	ADL AT %M*				: REAL := 1.0;		//Gräns konfliktlarm~wp:[unit]%
	AD AT %M*		 		: INT := 60;		//Larmfördröjning konfliktlarm~wp:[unit]s
END_VAR

	//Blockering handställning
	IF bInterlock THEN
		M := FALSE;
	END_IF;

	//Handställning
	IF M  THEN
		OP := OPM; 
	ELSE
		OP := rSetpoint;  
	END_IF
	
	//Handställningslarm
	fbAlarm2(bInput:=M , tAlarmDelay:= , bAutoReset:=TRUE , bAlarmOutput=>AL8 );
	
	//Invertering utång
	IF bInvert THEN
		rOutputInternal := (100 - OP);
	ELSE 
		rOutputInternal := OP;
	END_IF;		
		
	//Hantering utgång	
	FB_BA_AO01(
		rX:= rOutputInternal, 
		rX01:= 0, 
		rX02:= 100, 
		rY01:= 0, 
		rY02:= 32767 , 
		udiOpMod:= , 
		rXManual:= , 
		rY=> rY, 
		TO_iY=>TO_iY );
		
	//Hantering ingång (för feedback)
		FB_BA_AI01(
	TI_usiState:= usiState, 
	TI_iDataIn:= iDataIn, 
	eTerminal:= AIiBusTermType, 
	eSensor:= 0, (* 0 = pt1000, *)
	bConfigurate:= , 
	rX01:=AIrScaleX1 , 
	rX02:=AIrScaleX2 , 
	rY01:= AIrScaleMin, 
	rY02:= AIrScaleMax, 
	rOffset:= , 
	rSmoothingFactor:= , 
	udiDecimalPlace:= , 
	bEnLimitCtrl:= , 
	rHighLimit:= , 
	rLowLimit:=, 
	udiDelayLimitCtrl_sec:= , 
	TO_usiCtrl=> usiCtrl, 
	TO_iDataOut=> iDataOut, 
	rVal=> , 
	bWireBreak=> , 
	bShortCircuit=> , 
	bHighLimit=> , 
	bLowLimit=> , 
	bErr=> , 
	sErrDescr=> );
	
	FB_BA_TiAvrg01(
	bEn:= TRUE, 
	bEnAvrg := TRUE,
	lrIn:=REAL_TO_LREAL(FB_BA_AI01.rVal), 
	udiIntval:=1, 
	udiNumOfElem:= iMedelvardeSekunder, 
	lrOut=> );
	
	IF AI_M THEN
		PV := AI_OPM;
	ELSE
		PV := LREAL_TO_REAL(FB_BA_TiAvrg01.lrOut) + rCal;
	END_IF
	
FAULT := FB_BA_AI01.bWireBreak OR FB_BA_AI01.bShortCircuit;

//Konfliktlarm återföring; tillåt larmtimer om OP ej förändrats mer än tillåten avvikelse, larmvillkor om avvikelse OP-PV större än gräns
IF ABS(OP - rOPold) > ADL THEN
	fbAlarmFb.bInput := FALSE;
	rOPold := OP;
ELSE
	fbAlarmFb.bInput:= ABS(OP - PV) > ADL;
END_IF

fbAlarmFb(tAlarmDelay:= DINT_TO_TIME(AD) * 1000, bAutoReset:=TRUE , bAlarmOutput=>AL );

END_FUNCTION_BLOCK

// oaksLibrary/Utsignal DO_AO/fbComfoVent
//Hantering av vädringsluckor som är pulstidsstyrda med öppetindikering (ej stängt)
FUNCTION_BLOCK fbComfoVent
VAR_INPUT
	V1 AT %M*	: BOOL; //Kommando öppna läge 1 (delvis öppet) ~wp:[trendoptions]i:14400, t:1
	V2 AT %M*	: BOOL; //Kommando öppna läge 2 (fullt öppet) ~wp:[trendoptions]i:14400, t:1
	bInd : BOOL; //Öppetindikering;
END_VAR
VAR_OUTPUT
	bOppna	: BOOL; //Kommando öppna (till DO)
	bStang	: BOOL; //Kommando stäng (till DO)
	PV1 AT %M* : STRING(30); //Aktuellt läge ~wp:
	AL AT %M*	: BOOL; //Fel läge vädringsluckor~wp:
	AL8 AT %M* : BOOL; //Vädringsluckor ej i autoläge ~wp:
END_VAR
VAR
	fbPuls	: TON;
	bInit : BOOL := TRUE;
	
	fbEdge1, fbEdge2 : fbEdge;
	fbAlarm : fbAlarm;
	bStangInt : BOOL;
END_VAR

VAR_INPUT PERSISTENT
	SP1 AT %M* : UINT := 15; //Gångtid kommando läge 1 (delvis öppet) ~wp:[unit]s
	SP2 AT %M* : UINT := 30; //Gångtid kommando läge 2 (fullt  öppet) ~wp:[unit]s
	SP3 AT %M* : UINT := 40; //Gångtid kommando stängt~wp:[unit]s
	AD AT %M*	: UINT := 120; //Fördröjning larm fel läge~wp:[unit]s
	MCMD AT %M* : BYTE; //Handkörning (Auto, Stäng, Öppna delvis, Öppna helt)~wp:[trendoptions]i:14400, t:1
END_VAR

//Handkörning: 1 = Stäng, 2 = Öppna delvis, 3 = Öppna helt
IF MCMD = 1 THEN
	V1 := FALSE;
	V2 := FALSE;
ELSIF MCMD = 2 THEN
	V1 := TRUE;
	V2 := FALSE;
ELSIF MCMD = 3 THEN
	V1 := FALSE;
	V2 := TRUE;
END_IF

AL8 := MCMD <> 0;

//Kolla om något av ingående kommandon förändrats
fbEdge1(anyInput := V1);
fbEdge2(anyInput := V2);

fbPuls.IN := FALSE;

//Återställ puls
IF fbEdge1.bEdgeF OR fbEdge2.bEdgeF THEN
	fbPuls(IN := FALSE);
END_IF

//Om kommando förändrats eller vid uppstart, börja alltid med att stänga helt för att få stängt läge som utgångspunkt
IF fbEdge1.bEdgeSR OR fbEdge2.bEdgeSR OR bInit OR bStangInt THEN
	fbPuls.PT := UINT_TO_TIME(SP3) * 1000;
	fbPuls.IN := TRUE;
	bOppna := FALSE;
	bStang := NOT fbPuls.Q;
	
	IF fbPuls.Q AND NOT bInd THEN
		fbEdge1(bRst := TRUE);
		fbEdge2(bRst := TRUE);
		bInit := FALSE; 
		bStangInt := FALSE;
		fbPuls.IN := FALSE;
	END_IF
	
ELSE
	//Öppna delvis
	IF V1 THEN
		fbPuls.IN := TRUE;
		fbPuls.PT := UINT_TO_TIME(SP1) * 1000;
		bOppna := NOT fbPuls.Q;
	//Öppna helt 
	ELSIF V2 THEN
		fbPuls.IN := TRUE;
		fbPuls.PT := UINT_TO_TIME(SP2) * 1000;
		bOppna := NOT fbPuls.Q;
	END_IF;
END_IF;

fbPuls();

//Larm fel läge
fbAlarm(bInput := (V1 OR V2) XOR bInd, tAlarmDelay := DINT_TO_TIME(AD) * 1000, bAutoReset := TRUE, bAlarmOutput => AL);

//Sätt statustext
IF bStang THEN
	PV1 := 'Stänger';
ELSIF bOppna THEN
	PV1 := 'Öppnar';
ELSIF NOT (V1 OR V2) THEN
	PV1 := 'Stängt';
ELSIF V1 THEN
	PV1 := 'Delvis öppet';
ELSIF V2 THEN
	PV1 := 'Helt öppet';
END_IF;

END_FUNCTION_BLOCK

// oaksLibrary/Utsignal DO_AO/fbDigitalSignalLogicFb
//Block för digitala utsignaler med möjlighet att handställa utsignal. Larmar vid handställning.
//Ingång för lägesåterföring (feedback) för visning samt generering av larm om konflikt mellan M och V0/V1 (feedback)
FUNCTION_BLOCK fbDigitalSignalLogicFb
VAR_INPUT
	bStart : BOOL; //startvillkor
	bSafe: BOOL; //Säkerhetsvillkor
	bHandsetBlock : BOOL; //Används för blockering av handställning utan att blockera utsignal i autoläge. OBS! - För säkerhetsvillkor se ingång bSafe!
	tStartDelay : TIME := T#0S; //Startfördröjning
	tStopDelay : TIME := T#0S; //Stoppfördröjning
	
	V0 AT %I* : BOOL; //Indikering stängd~wp:[trendoptions]i:14400, t:1
	V1 AT %I* : BOOL; //Indikering öppen~wp:[trendoptions]i:14400, t:1
END_VAR
VAR_OUTPUT
	{attribute 'OPC.UA.DA' := '1'}
	CMD AT %Q* 			: BOOL; 		//Utsignal~wp:[trendoptions]i:300[trendoptions]i:14400, t:1
	{attribute 'OPC.UA.DA' := '1'}
	AL8 AT %M* 			: BOOL; 		//Utsignal handställd~wp:[alarmoptions]p:3
	STATE1 AT %M* 		: STRING; 		//Status IO-modul~wp:
	tStartDelayRemaining: TIME; 		//Aktuell  återstående tid startfördröjning
	tStopDelayRemaining : TIME; 		//Aktuell återstående tid toppfördröjning
	AL AT %M* 			: BOOL;			//Konfliktlarm~wp:[alarmoptions]p:3
END_VAR
VAR
	bInternalStart 		: BOOL;
	fbAlarm2 			: fbAlarm; //Larm handställning
	fbAlarmFb			: fbAlarm; //Konfliktlarm
	//Handställningsvariabler från IO
	TI_bStateAuto AT %I* 	:BOOL :=TRUE; //Status Auto/Manuell
	TI_bStateRelay AT %I* 	:BOOL :=FALSE; //Status reläutgång
	bIOManual 				: BOOL;
	
	fbStartDelay	: TON; //Startfördröjning
	fbStopDelay		: TOF; //Stoppfördröjning
END_VAR
VAR_INPUT PERSISTENT
	{attribute 'OPC.UA.DA' := '1'}
	M AT %M* 	: BOOL; //Handställning~wp:[trendoptions]i:14400, t:1
	{attribute 'OPC.UA.DA' := '1'}
	MCMD AT %M* : BOOL; //Styrsignal handställning~wp:[trendoptions]i:14400, t:1
	
	AD AT %M* 	: INT := 60; //Larmfördröjning konfliktlarm~wp:[unit]s
END_VAR

	//Handställning
	fbAlarm2(bInput:=M OR NOT TI_bStateAuto, tAlarmDelay:= , bAutoReset:=TRUE , bAlarmOutput=>AL8 );
	
	IF NOT bSafe OR bHandsetBlock THEN
		M := FALSE;
	END_IF;
	
	//Manuell omkopplare IO-modul
	bIOManual := fKx2652State(bAuto := TI_bStateAuto, bRelayStatus := TI_bStateRelay, sState => STATE1);
	
	
	//Start-/stoppfördröjning
    fbStartDelay(IN:=bStart , PT:=tStartDelay , Q=> , ET=> );
	fbStopDelay(IN:=fbStartDelay.Q, PT:=tStopDelay , Q=> , ET=> );
	
	tStopDelayRemaining := mTimeRemainingTof(fbStopDelay);
	tStartDelayRemaining := mTimeRemainingTon(fbStartDelay);
	
	bInternalStart := fbStopDelay.Q;
	
	IF NOT TI_bStateAuto THEN
		CMD := bIOManual;
	ELSE
		CMD := (((bInternalStart AND NOT M) OR (M AND MCMD)) AND bSafe) OR bIOManual;
	END_IF
	
//Konfliktlarm återföring
fbAlarmFb(
	bInput:= (CMD AND NOT V1) OR (CMD AND V0) OR (NOT CMD AND V1) OR (NOT CMD AND NOT V0), 
	tAlarmDelay:= DINT_TO_TIME(AD) * 1000, 
	bAutoReset:=TRUE, 
	bAlarmOutput=>AL
);

METHOD PUBLIC mStartDelayRemaining : STRING
VAR_INPUT
	sStatusString : STRING;
END_VAR
VAR
	tTime : TIME; 
END_VAR
	tTime := mTimeRemainingTon(fbStartDelay);
	
	
	IF tTime > T#0S AND tTime < fbStartDelay.PT AND NOT M AND TI_bStateAuto  THEN
 		mStartDelayRemaining := CONCAT(sStatusString,CONCAT(INT_TO_STRING(TIME_TO_INT(tTime/1000)), ' s'));
	ELSE
		mStartDelayRemaining := ' ';
	END_IF
END_METHOD

METHOD PUBLIC mStopDelayRemaining : STRING
VAR_INPUT
	sStatusString : STRING;
END_VAR
VAR
	tTime : TIME; 
END_VAR
	tTime := mTimeRemainingTof(fbStopDelay);
	
	
	IF tTime > T#0S AND tTime < fbStopDelay.PT AND NOT M AND TI_bStateAuto  THEN
 		mStopDelayRemaining := CONCAT(sStatusString,CONCAT(INT_TO_STRING(TIME_TO_INT(tTime/1000)), ' s'));
	ELSE
		mStopDelayRemaining := ' ';
	END_IF
END_METHOD

METHOD PROTECTED mTimeRemainingTof : TIME
VAR_IN_OUT
	fbTof : TOF;
END_VAR
mTimeRemainingTof := fbTof.PT - fbTof.ET;
END_METHOD

METHOD PROTECTED mTimeRemainingTon : TIME
VAR_IN_OUT
	fbTon : TON;
END_VAR
mTimeRemainingTon := fbTon.PT - fbTon.ET;
END_METHOD

END_FUNCTION_BLOCK

// oaksLibrary/Utsignal DO_AO/fbGeneralSignalLogic
//OAKS AB
//2022-10-28
//Generellt analog ut block med handställningsmöjlighet för tex. ventilställdon via SX:Acura
FUNCTION_BLOCK fbGeneralSignalLogic
VAR_INPUT
	rSetpoint 				: REAL := 0; //Skalad insignal för auto-läge (exmepelvis regulatorsignal)
	bInterlock 				: BOOL := FALSE; //Blockering av handställning
	bInvert 				: BOOL := FALSE; //Invertering utgång
END_VAR
VAR_OUTPUT
	{attribute 'OPC.UA.DA' := '1'}
	AL8 AT %M* 				: BOOL := FALSE; //Utsignal handställd~wp:[alarmoptions]p:3
	{attribute 'OPC.UA.DA' := '1'}
	OP AT %M* : REAL;  //Utsignal~wp:[unit]%[format]0[trendoptions]i:300
END_VAR
VAR
	rOutputInternal 		: REAL; //Intern signal för invertering/ej invertering
	rOutputConverted		: REAL; //Signal inverterad eller/ej inverterad
	fbAlarm2 				: fbAlarm; //Larm handställning
END_VAR
VAR_INPUT PERSISTENT
	{attribute 'OPC.UA.DA' := '1'}
	M AT %M*				: BOOL;//Handställning~wp:[trendoptions]i:14400, t:1
	{attribute 'OPC.UA.DA' := '1'}
	OPM AT %M* : REAL;//Värde handställning~wp:[unit]%[format]0
END_VAR

	//Blockering handställning
	IF bInterlock THEN
		M := FALSE;
	END_IF;

	//Handställning
	IF M THEN
		rOutputConverted := OPM; 
	ELSE
		rOutputConverted := rSetpoint;  
	END_IF
	
	//Handställningslarm
	fbAlarm2(bInput:=M , tAlarmDelay:= , bAutoReset:=TRUE , bAlarmOutput=>AL8 );
	
	//Invertering utång
	IF bInvert THEN
		rOutputInternal := (100 - rOutputConverted);
	ELSE 
		rOutputInternal := rOutputConverted;
	END_IF;		

	//Utsignal 
	OP := rOutputInternal;

END_FUNCTION_BLOCK

// oaksLibrary/Utsignal DO_AO/fbLightSignalLogic
// Funktionsblock för utebelysning ute. Valbart driftläge för startvillkor mellan Astrour + Tidkanal och enbart Tidkanal.
// ANVÄND EJ bStart då denna skrivs till internt i blocket.
FUNCTION_BLOCK fbLightSignalLogic EXTENDS fbDigitalSignalLogic
VAR_INPUT
	bTidkanal : BOOL; // Koppla tidkanal hit.
	bAstrour : BOOL; // Koppla utgång från fbSunclock hit.
END_VAR
VAR_OUTPUT
END_VAR
VAR
END_VAR
VAR PERSISTENT
	{attribute 'OPC.UA.DA' := '1'}
	SP1 AT %M* : INT; //1 = Astrour + Tidkanal. 0 = Tidkanal~wp:
END_VAR	
VAR_OUTPUT
	{attribute 'OPC.UA.DA' := '1'}
	PV AT %M* : STRING; //Startvillkor~wp:
END_VAR

SUPER^();
bStart := mBelysningsvillkor(iDriftlage:= SP1, bTidkanal:=bTidkanal , bAstrour:= bAstrour, sAktuelltDriftlage=>PV);

METHOD PRIVATE mBelysningsvillkor : BOOL
VAR_IN_OUT
	iDriftlage : INT; // 1 om belysningsvillkor OCH tidkanal måste vara till. 0 om bara tidkanal måste vara till.
END_VAR
VAR_INPUT
	bTidkanal : BOOL;
	bAstrour : BOOL; // lux-givare under inställt värde
END_VAR
VAR_OUTPUT
	sAktuelltDriftlage : STRING;
END_VAR
IF bTidkanal AND bAstrour THEN
	mBelysningsvillkor := TRUE;
ELSIF bTidkanal AND iDriftlage = 0 THEN
	mBelysningsvillkor := TRUE;
ELSE
	mBelysningsvillkor := FALSE;
END_IF

IF iDriftlage = 1 THEN
	sAktuelltDriftlage := 'Tidkanal och astrour sätter utgång i läge till.';
ELSE
	sAktuelltDriftlage := 'Tidkanal sätter utgång i läge till.';
END_IF

IF iDriftlage > 1 THEN
	iDriftlage := 1; 
END_IF

IF iDriftlage < 0 THEN
	iDriftlage := 0; 
END_IF
END_METHOD

END_FUNCTION_BLOCK

// oaksLibrary/Utsignal DO_AO/fbLightSignalLogicLux
//Oaks AB
//2022-08-17
//Funktionsblock för utebelysning ute. Valbart driftläge för startvillkor mellan Luxgivare + Tidkanal och enbart Tidkanal.
//ANVÄND EJ bStart då denna skrivs till internt i blocket
FUNCTION_BLOCK fbLightSignalLogicLux EXTENDS fbDigitalSignalLogic
VAR_INPUT
	//Koppla tidkanal hit.
	bTidkanal: BOOL;
	//Koppla utgång från LuxLightCon blocket hit eller egen hyst hit.
	bLux: BOOL;
END_VAR
VAR PERSISTENT
	//1 = Luxgivare + Tidkanal. 0 = Tidkanal~wp:
	{attribute 'OPC.UA.DA' := '1'}
	SP1 AT %M*: INT;
END_VAR
VAR_OUTPUT
	//Startvillkor~wp:
	{attribute 'OPC.UA.DA' := '1'}
	PV AT %M*: STRING;
END_VAR

SUPER^();
bStart := mBelysningsvillkor(iDriftlage:= SP1, bTidkanal:=bTidkanal , bLux:= bLux, sAktuelltDriftlage=>PV);

METHOD mBelysningsvillkor : BOOL
VAR_IN_OUT
	/// 1 om belysningsvillkor OCH tidkanal måste vara till. 0 om bara tidkanal måste vara till.
	iDriftlage: INT;
END_VAR
VAR_INPUT
	bTidkanal: BOOL;
	/// lux-givare under inställt värde
	bLux: BOOL;
END_VAR
VAR_OUTPUT
	sAktuelltDriftlage: STRING;
END_VAR
IF bTidkanal AND bLux THEN
	mBelysningsvillkor := TRUE;
ELSIF bTidkanal AND iDriftlage = 0 THEN
	mBelysningsvillkor := TRUE;
ELSE
	mBelysningsvillkor := FALSE;
END_IF

IF iDriftlage = 1 THEN
	sAktuelltDriftlage := 'Tidkanal och luxgivare sätter utgång i läge till.';
ELSE
	sAktuelltDriftlage := 'Tidkanal sätter utgång i läge till.';
END_IF

IF iDriftlage > 1 THEN
	iDriftlage := 1; 
END_IF

IF iDriftlage < 0 THEN
	iDriftlage := 0; 
END_IF
END_METHOD

END_FUNCTION_BLOCK

// oaksLibrary/Växlingsblock/fbDailyToggle
// Block för att växla mellan två bool-outputs. Växling sker intälld tid varje dag.
FUNCTION_BLOCK fbDailyToggle
VAR_INPUT
	{attribute 'OPC.UA.DA' := '1'}
	M AT %M*  : BOOL; //Manuell växling~wp:[trendoptions]i:14400, t:1
END_VAR
VAR_OUTPUT
	{attribute 'OPC.UA.DA' := '1'}
	PV AT %M* : INT; //Aktuellt val~wp:[trendoptions]i:14400, t:1
	bOutput1, bOutput2 : BOOL;
END_VAR
VAR 
	fbDayTrig: R_trig;
	{attribute 'OPC.UA.DA' := '1'}
	PV4 AT %M* : STRING := ' ' ; //Växling sker intälld tid varje dag. Tiden är ställbar mellan 0000-2359.~wp:
	stTime		: tc2_ba.TIMESTRUCT;
	nActualDayCase	: INT;
	nActualHour 	: INT;
	nActualMinute 	: INT;
	
	FB_BA_GetTime01 : tc2_ba.FB_BA_GetTime; 
	FB_BA_ExtTiSt01 : tc2_ba.FB_BA_ExtTiSt;	
	
	nTime : INT; // Internvariabel aktuell tid (nActualHour+nActualMinute)
//	bDay : BOOL; // Internvariabel blir TRUE om inställd dag är lika med aktuell dag
	bTime : BOOL; // Internvariabel blir TRUE om inställd tid är lika med aktuell tid
END_VAR
VAR_INPUT PERSISTENT
//	SP1 AT %M*  : INT:=1; //Dag för växling (-1 = ingen växling 0 = Söndag 1 = Måndag 2 = Tisdag..7 = Söndag~wp:
	{attribute 'OPC.UA.DA' := '1'}
	SP1 AT %M*  : INT:=1000; //Tid för växling (skrivs i format 1200 för 12:00)~wp:
END_VAR

	FB_BA_GetTime01(bEn :=TRUE);	
	stTime := FB_BA_GetTime01.stSysTi;

//	nActualDayCase :=WORD_TO_INT (stTime.wDayOfWeek);
	nActualHour :=WORD_TO_INT (stTime.wHour)*100;
	nActualMinute :=WORD_TO_INT (stTime.wMinute);
	
	nTime := nActualHour+nActualMinute;
	
//	bDay := nActualDayCase = SP1;
	bTime := nTime = SP1;

//	IF SP1 < -1 OR  SP1>7 THEN
//		SP1 := 1;
//	END_IF
	
	IF SP1 < 0 OR  SP1>2359 THEN
		SP1 := 1200;
	END_IF

	IF PV < 1 OR PV > 2  THEN	
		PV := 1;
	END_IF;

	IF bTime OR M THEN
		fbDayTrig(CLK := TRUE);
	ELSE
		fbDayTrig(CLK := FALSE);
	END_IF

	IF fbDayTrig.Q THEN
		IF PV = 1 THEN
			PV := 2;
		ELSE
			PV := 1;
		END_IF
	END_IF
	
	bOutput1 := (PV = 1);
	bOutput2 := (PV = 2);

END_FUNCTION_BLOCK

// oaksLibrary/Växlingsblock/fbMonthlyToggle
// Block för att växla mellan två bool-outputs. Växling sker intälld tid på inställd dag (-1 till 31).
FUNCTION_BLOCK fbMonthlyToggle
VAR_INPUT
	{attribute 'OPC.UA.DA' := '1'}
	M AT %M*  : BOOL; //Manuell växling~wp:[trendoptions]i:14400, t:1
END_VAR
VAR_OUTPUT
	{attribute 'OPC.UA.DA' := '1'}
	PV AT %M* : INT; //Aktuellt val~wp:[trendoptions]i:14400, t:1
	bOutput1, bOutput2 : BOOL;
END_VAR
VAR 
	fbDayTrig: R_trig;
	{attribute 'OPC.UA.DA' := '1'}
	PV4 AT %M* : STRING := ' ' ; //Växling sker intälld tid på inställd dag (1-31). Ställer man in -1 på "Dag för växling" så inaktiveras växlingen. Tänk på att alla månader inte har 31 dagar. Tiden är ställbar mellan 0000-2359.~wp:
	stTime		: tc2_ba.TIMESTRUCT;
	nActualDayCase	: INT;
	nActualHour 	: INT;
	nActualMinute 	: INT;
	
	FB_BA_GetTime01 : tc2_ba.FB_BA_GetTime; 
	FB_BA_ExtTiSt01 : tc2_ba.FB_BA_ExtTiSt;	
	
	nTime : INT; // Internvariabel aktuell tid (nActualHour+nActualMinute)
	bDay : BOOL; // Internvariabel blir TRUE om inställd dag är lika med aktuell dag
	bTime : BOOL; // Internvariabel blir TRUE om inställd tid är lika med aktuell tid
END_VAR
VAR_INPUT PERSISTENT
	{attribute 'OPC.UA.DA' := '1'}
	SP1 AT %M*  : INT:=1; //Dag för växling (1-31)~wp:
	{attribute 'OPC.UA.DA' := '1'}
	SP2 AT %M*  : INT:=1000; //Tid för växling (skrivs i format 1200 för 12:00)~wp:
END_VAR

	FB_BA_GetTime01(bEn :=TRUE);	
	stTime := FB_BA_GetTime01.stSysTi;

	nActualDayCase :=WORD_TO_INT (stTime.wDay);
	nActualHour :=WORD_TO_INT (stTime.wHour)*100;
	nActualMinute :=WORD_TO_INT (stTime.wMinute);
	
	nTime := nActualHour+nActualMinute;
	
	bDay := nActualDayCase = SP1;
	bTime := nTime = SP2;

	IF SP1 < -1 OR  SP1>31 THEN
		SP1 := 1;
	END_IF
	
	IF SP2 < 0 OR  SP2>2359 THEN
		SP2 := 1200;
	END_IF

	IF PV < 1 OR PV > 2  THEN	
		PV := 1;
	END_IF;

	IF (bDay AND bTime) OR M THEN
		fbDayTrig(CLK := TRUE);
	ELSE
		fbDayTrig(CLK := FALSE);
	END_IF

	IF fbDayTrig.Q THEN
		IF PV = 1 THEN
			PV := 2;
		ELSE
			PV := 1;
		END_IF
	END_IF
	
	bOutput1 := (PV = 1);
	bOutput2 := (PV = 2);

END_FUNCTION_BLOCK

// oaksLibrary/Växlingsblock/fbToggleStep
// Toggle-funktion med uppstegning. Togglar abOutput[0..9] (eller max inst.) i sekvens med inställt intervall när bStart är till.
FUNCTION_BLOCK fbToggleStep
VAR_INPUT
	bStart 		: BOOL;
	iMaxStep	: INT := 9;
	tTimeOn 	: TIME := T#10S;
	tTimeOff 	: TIME := T#10S;
	
END_VAR
VAR_OUTPUT
	iStep		: INT := 0;
	abOutput 	: ARRAY[0..9] OF BOOL;
END_VAR
VAR	
	fbTrigger 	: r_trig;
	fbTon1 		: ton;
	fbTof2 		: tof;
	iX			: INT;
END_VAR

IF iMaxStep > 9 THEN
	iMaxStep := 9;
END_IF

IF bStart THEN
	fbTon1(IN:= NOT fbTof2.Q, PT:= tTimeOff , Q=> , ET=> );
	
	IF fbTon1.Q THEN
		fbTrigger(CLK:=TRUE , Q=> );
		fbTof2(IN:=fbTrigger.Q , PT:=tTimeOn , Q=> , ET=> );
	ELSE
		fbTof2(IN:=FALSE , PT:=tTimeOn , Q=> , ET=> );
		fbTrigger(CLK:=FALSE , Q=> );		
	END_IF
	
	IF fbTrigger.Q THEN
		iStep := iStep + 1;
		IF iStep > iMaxStep THEN
			iStep := 0;
		END_IF
	END_IF
	
	FOR iX := 0 TO 9 DO 
		abOutput[iX] := (iStep = iX) AND fbTof2.Q;
	END_FOR;
ELSE
	FOR iX := 0 TO 9 DO 
		abOutput[iX] := FALSE;
	END_FOR;
END_IF
fbTof2();
fbTon1();

END_FUNCTION_BLOCK

// oaksLibrary/Växlingsblock/fbWeeklyToggle
// Block för att växla mellan två bool-outputs. Växling sker intälld tid på inställd veckodag (-1 till 7).
FUNCTION_BLOCK fbWeeklyToggle
VAR_INPUT
	{attribute 'OPC.UA.DA' := '1'}
	M AT %M*  : BOOL; //Manuell växling~wp:[trendoptions]i:14400, t:1
END_VAR
VAR_OUTPUT
	{attribute 'OPC.UA.DA' := '1'}
	PV AT %M* : INT; //Aktuellt val~wp:[trendoptions]i:14400, t:1
	bOutput1, bOutput2 : BOOL;
END_VAR
VAR 
	fbDayTrig: R_trig;
	{attribute 'OPC.UA.DA' := '1'}
	PV4 AT %M* : STRING := ' ' ; //Växling sker intälld tid på inställd veckodag. Ställer man in -1 på "Dag för växling" så inaktiveras växlingen. Tiden är ställbar mellan 0000-2359.~wp:
	stTime		: tc2_ba.TIMESTRUCT;
	nActualDayCase	: INT;
	nActualHour 	: INT;
	nActualMinute 	: INT;
	
	FB_BA_GetTime01 : tc2_ba.FB_BA_GetTime; 
	FB_BA_ExtTiSt01 : tc2_ba.FB_BA_ExtTiSt;	
	
	nTime : INT; // Internvariabel aktuell tid (nActualHour+nActualMinute)
	bDay : BOOL; // Internvariabel blir TRUE om inställd dag är lika med aktuell dag
	bTime : BOOL; // Internvariabel blir TRUE om inställd tid är lika med aktuell tid
END_VAR
VAR_INPUT PERSISTENT
	{attribute 'OPC.UA.DA' := '1'}
	SP1 AT %M*  : INT:=1; //Dag för växling (0 = Söndag 1 = Måndag 2 = Tisdag..7 = Söndag)~wp:
	{attribute 'OPC.UA.DA' := '1'}
	SP2 AT %M*  : INT:=1000; //Tid för växling (skrivs i format 1200 för 12:00)~wp:
END_VAR

	FB_BA_GetTime01(bEn :=TRUE);	
	stTime := FB_BA_GetTime01.stSysTi;

	nActualDayCase :=WORD_TO_INT (stTime.wDayOfWeek);
	nActualHour :=WORD_TO_INT (stTime.wHour)*100;
	nActualMinute :=WORD_TO_INT (stTime.wMinute);
	
	nTime := nActualHour+nActualMinute;
	
	bDay := nActualDayCase = SP1;
	bTime := nTime = SP2;

	IF SP1 < -1 OR  SP1>7 THEN
		SP1 := 1;
	END_IF
	
	IF SP2 < 0 OR  SP2>2359 THEN
		SP2 := 1200;
	END_IF

	IF PV < 1 OR PV > 2  THEN	
		PV := 1;
	END_IF;

	IF (bDay AND bTime) OR M THEN
		fbDayTrig(CLK := TRUE);
	ELSE
		fbDayTrig(CLK := FALSE);
	END_IF

	IF fbDayTrig.Q THEN
		IF PV = 1 THEN
			PV := 2;
		ELSE
			PV := 1;
		END_IF
	END_IF
	
	bOutput1 := (PV = 1);
	bOutput2 := (PV = 2);

END_FUNCTION_BLOCK

// oaksLibrary/fbExcerciseInactiveMotor
FUNCTION_BLOCK fbExcerciseInactiveMotor		//Funktionsblock för att motionera en komponent efter att den ej körts under viss tid
VAR_INPUT
	bRunIndication	: BOOL;		//Ska vara till när komponenten går (t ex driftsvar)
	tInactiveTime	: TIME;		//Tid som skall passera utan att komponenten går till för att motion skall ske
	tExcerciseTime	: TIME;		//Gångtid motionskörning
END_VAR

VAR
	fbTON			: TON;		//Timer som startar motion
	fbTOF			: TOF;		//Timer för motionering
END_VAR

VAR_OUTPUT
	bOutput			: BOOL;		//Motioneringskommando
	tTimeLeftNext	: TIME;		//Tid kvar till nästa motion
	tTimeLeftExc	: TIME;		//Tid kvar motionering
END_VAR

//Kör TON med inställd tid när komponenten inte går
fbTON(IN := NOT bRunIndication, PT := tInactiveTime);

//Kör TOF med inställd tid när TON gått till, dvs motionering ska starta, skriv utsignal
fbTOF(IN := fbTON.Q, PT := tExcerciseTime, Q => bOutput);	

tTimeLeftNext 	:= tInactiveTime - fbTON.ET;
tTimeLeftExc	:= tExcerciseTime - fbTOF.ET;

END_FUNCTION_BLOCK

// oaksLibrary/fbNightCooling
FUNCTION_BLOCK fbNightCooling
// Funktionsblock för nattkyla
// Ändrat av Robert H, 2021-11-23
// Testat 2021-11-23

// V-tagg i detta block knyts till regulator för att blockera eventuell kylsekvens, till inputen bNightCooling i fbVentilationUnit.
VAR
	fbExhTemperatureTON : TON;
	rLocalTemperatureProcessValue : REAL; // Mellanvariabel för temperatur. Vid nattkyla via frånluftstemperatur uppdateras denna enbart vid driftindikering på frånluftsfläkt.
	summerInternal: BOOL;
	bNightCool : BOOL;
	fbTof_StopDelayNC: TOF;
	fbTon_StartDelaySummer: TON;
	fbTof_StopDelaySummer: TOF;
	sTemp : STRING(255);
	rTempUsed : REAL; // Uteluftstemperatur
END_VAR

VAR_INPUT
	bExhfanInd : BOOL; // Vid nattkyla via frånluftstemp knyt frånluftsfläktens indikering.
	bExhtempMode : BOOL; // Aktivera denna för nattkyla via frånluftstemp.
	rSetpoint : REAL; // Börvärde. Knyt det börvärde som används vid normaldrift (exempelvis utekomp eller kaskad).	
	bTimechannel : BOOL; //Dagdrift (knyt outputen bNormalOperation från fbVentilationUnit)	
	rOutdoorTemperature : ANY; //Utetemperatur knyter man inget här används oaksGVL.rOutdoortemp
END_VAR
VAR_INPUT PERSISTENT
	Enable : BOOL := TRUE; // Tillåt nattkyla (knyt t ex _M-tagg eller villkor från annan funktion)
	{attribute 'OPC.UA.DA' := '1'}
	PV AT %M*  : REAL; //Aktuell temperatur~wp:[unit]°C[format]0.0
	{attribute 'OPC.UA.DA' := '1'}
	SP AT %M*  : REAL := 22; //Rumsbörvärde nattkyla (startar 2.5°C över och stoppar 0.5°C under~wp:[unit]°C[format]0.0
	{attribute 'OPC.UA.DA' := '1'}
	SP1 AT %M*  : REAL := 14; //Börvärde tilluft vid nattkyla~wp:[unit]°C[format]0.0
	{attribute 'OPC.UA.DA' := '1'}
	SP2 AT %M*  : REAL := 12; //Mingräns utetemp för nattkyla~wp:[unit]°C[format]0.0
END_VAR

VAR_OUTPUT
	{attribute 'OPC.UA.DA' := '1'}
	V AT %M* : BOOL; //Nattkyla aktiv~wp:[trendoptions]i:14400, t:1
	{attribute 'OPC.UA.DA' := '1'}
	PV4 AT %M*  : BOOL; // Startvillkor rumstemperatur över~wp:[trendoptions]i:14400, t:1
	{attribute 'OPC.UA.DA' := '1'}
	PV5 AT %M* : BOOL; //Utetemperaturvillkor nattkyla~wp:[trendoptions]i:14400, t:1
	{attribute 'OPC.UA.DA' := '1'}
	PV6 AT %M*  : BOOL; // Startvillkor rumstemperatur högre än utetemp~wp:[trendoptions]i:14400, t:1
	{attribute 'OPC.UA.DA' := '1'}
	PV7 AT %M*  : STRING; // Konfiguration nattkyla~wp:
	{attribute 'OPC.UA.DA' := '1'}
	PV8 AT %M*  : STRING; // Konfiguration nattkyla~wp:
	rSetpointOutput : REAL; // Aktuellt börvärde. Knyts till CSP tilluft (använder man våra setpoint-block knyter man denna till rOverrideSetpoint)
END_VAR

//Temp select
	rTempUsed := F_GetTempToUse(rOutdoorTemperature);

	sTemp := 'Nattkyla via: ';
	IF bExhtempMode THEN
		sTemp := CONCAT(sTemp, 'Frånluftstemperatur');
	ELSE
		sTemp := CONCAT(sTemp, 'Rumstemperatur');	
	END_IF
		
	PV7 := sTemp;
	
	sTemp := 'Aktuell nattkyletemperatur: ';
	
	sTemp := CONCAT(sTemp, REAL_TO_STRING(rLocalTemperatureProcessValue));	
	PV8 :=CONCAT(sTemp, ' °C');
	//Summer	
	IF (rTempUsed > SP2) AND Enable THEN
		summerInternal := TRUE;
	ELSIF (rTempUsed < (SP2 - 0.5)) OR NOT Enable THEN
		summerInternal := FALSE;
	END_IF;
	
	//Start/stop delay summer
   	fbTon_StartDelaySummer(IN:= summerInternal, PT:= T#15M, Q=>, ET=> );
	fbTof_StopDelaySummer(IN:= fbTon_StartDelaySummer.Q, PT:= T#5M, Q=>, ET=> );

	PV5 := fbTon_StartDelaySummer.Q OR fbTof_StopDelaySummer.Q;
	
	
	fbExhTemperatureTON(IN:=bExhfanInd , PT:=T#1M , Q=> , ET=> );
	
	IF fbExhTemperatureTON.Q OR NOT bExhtempMode THEN
		rLocalTemperatureProcessValue := PV;
	END_IF;
	
	IF rLocalTemperatureProcessValue > (SP + 2.5) THEN
		PV4 := TRUE;
	ELSIF rLocalTemperatureProcessValue < (SP - 0.5) THEN
		PV4 := FALSE;
	END_IF
	
	IF rTempUsed < (rLocalTemperatureProcessValue - 4.0) THEN
		PV6 := TRUE;
	ELSIF (rLocalTemperatureProcessValue - rTempUsed) < 3.0 THEN
		PV6 := FALSE;
	END_IF
	
	//Start/stop nightcool
	IF PV4 AND PV6 AND PV5 THEN
		bNightCool := TRUE;
	END_IF
	IF NOT PV4 OR NOT PV6 OR NOT PV5 THEN 
		bNightCool := FALSE;
	END_IF
	
	//Start/stop delay		
	fbTof_StopDelayNC(IN:= bNightCool, PT:= T#5M, Q=>, ET=> );
		
	V := fbTof_StopDelayNC.Q AND NOT bTimechannel;
		

	IF V THEN
		rSetpointOutput := SP1;
	ELSE
		rSetpointOutput := rSetpoint;
	END_IF

END_FUNCTION_BLOCK

// oaksLibrary/fbVentilationUnit
// Block för ventilationsaggregat. Förreglar aggregat vid Frysvakt, Driftfel, Brandlarm, Rökdetektorlarm, utlöst automatsäkring eller övriga förreglingar med möjlighet att sätta egen statustext.
// PV1 och PV2 indikerar ventilationsaggregatets aktuella status. 
FUNCTION_BLOCK fbVentilationUnit
VAR_INPUT
	bSequenceStart : BOOL := TRUE; // Vid sekvensstart knyt global variabel oaksgvl.bSekvensstart1-15 hit. Aggregat blockeras från att starta då denna ingång är FALSE.
	bServiceSwitch : BOOL; // Ingång serviceomkopplare
	bTimechannel : BOOL; // Startvillkor tidkanal
	bExtendedOperation : BOOL; // Startvillkor förlängd drift
	bUserDefinedOperation1 : BOOL; // Startvillkor egendefinierad drift
	sUserDefinedOperation1 : STRING :=  ' '; // Statustext vid egendefinierad drift (bUserDefinedOperation1)
	bUserDefinedOperation2 : BOOL; // Startvillkor egendefinierad drift
	sUserDefinedOperation2 : STRING :=  ' '; // Statustext vid egendefinierad drift (bUserDefinedOperation2)
	bNightCooling : BOOL; // Startvillkor nattkyla (används bara för statustext)
	bNightHeating : BOOL; // Startvillkor nattanvärmning (används bara för statustext)
	bCoolRecycling : BOOL; // Ingång kylåtervinning aggregat (används bara för statustext)
	bDefrostingVvx : BOOL; // Ingång avfrostning vvx (används bara för statustext)
	bFiredamperExercise : BOOL; // Stannar aggregatet och visar statustext. Aggregat återgår till drift efteråt. 
(*förreglingar - stänger ner aggregatet samt blockerar handställning *)
	bFreezeAlarm : BOOL; // Frysvakt
	bPumpAlarm : BOOL; // Driftfel pump värme
	bFireAlarm : BOOL; // Brandlarm
	bSmokeAlarm : BOOL; // Rökdetektorlarm
	bFuseAlarm : BOOL; // Förregling utlöst automatsäkring
	bInterlock : BOOL; // Övrig förregling
	sInterlockDescription : STRING :=  ' '; // Beskrivning för övrig förregling. Text visas i statusfält vid utlöst förregling
	bInterlock2 : BOOL; // Övrig förregling
	sInterlock2Description : STRING :=  ' '; // Beskrivning för övrig förregling. Text visas i statusfält vid utlöst förregling
	bInterlock3 : BOOL; // Övrig förregling
	sInterlock3Description : STRING :=  ' '; // Beskrivning för övrig förregling. Text visas i statusfält vid utlöst förregling
	
	tSupfanStartDelay : TIME := T#45S;
	tExhfanStartDelay : TIME := T#45S;
	
	tDamperStopDelay : TIME := T#10S; 	
	tAfterblowStopDelay : TIME := T#0S; // Efterblåsningstid vid elbatteri. Används för att köra tilluftsfläkten i angiven tid efter aggregatsstopp. !! Denna tidsinställning används även som stoppfördröjning för serviceomkopplare !!
	bAfterblowActive : BOOL := TRUE; // Knyt signal som indikerar att elbatteriet är aktivt. Efterblåsning i inställd tid körs om denna är true. Lämnas denna input tom körs efterblåsning alltid i inställd tid. 
	bSupfan_M : BOOL;
	bSupfan_MCMD : BOOL;
	bSupfanAlarm : BOOL;
	
	bExhfan_M : BOOL;
	bExhfan_MCMD : BOOL;
	bExhfanAlarm : BOOL;
END_VAR
VAR_OUTPUT
	bSupfanOutput : BOOL;
	bSupDamperOutput : BOOL;
	bExhfanOutput : BOOL;
	bExhDamperOutput : BOOL;
	
	bNormalOperation : BOOL; // Är till om aggregatet är i normaldrift (tidkanal eller förlängd drift)
	bNightHeatingStatus : BOOL; // Driftstatus nattanvärmning (Används för eventuell spjällstyrning va exempelvis återluft)
	bAfterBlowElectricHeaterStatus : BOOL; // Driftstatus efterblåsning elbatteri (Används för att blockera elbatteri-sekvens i regulator).
	bSafeCon : BOOL; // Säkerhetsvillkor 
	{attribute 'OPC.UA.DA' := '1'}
	PV1 AT %M* : STRING := ''; //Status aggregatsdrift~wp:[trendoptions]i:14400, t:1
	{attribute 'OPC.UA.DA' := '1'}
	PV2 AT %M* : STRING := ''; //Status aggregatsdrift~wp:[trendoptions]i:14400, t:1
	FAULT AT %M* : BOOL; //Larm lång drifttid~wp:[alarmoptions]p:3
END_VAR
VAR
	PV4 AT %M* : STRING; //Status drifttid~wp:[trendoptions]i:14400, t:1
	{attribute 'OPC.UA.DA' := '1'}
	PV9 AT %M* : BOOL; //Aktivt larm (används för portlet)~wp:[trendoptions]i:14400, t:1
	fbNattAnvarmningsFtrig : f_trig; // Blockerar normaldrift så att aggregat startar upp på nytt efter nattanvärmning
	fbNattAnvarmningsTof : TOF; //  Blockerar normaldrift så att aggregat startar upp på nytt efter nattanvärmning 
	fbInterlockAlarm : fbAlarm;
	bStartCon : BOOL; // Internvariabel startvillkor
	bStartConWithoutAfterblow : BOOL; // Internvariabel startvillkor utan efterblåsningsvillkor
	bExhfanCon : BOOL;
	bCrosswiseInterlock : BOOL;  // korsvis förregling
	
	bExhDamperCon : BOOL;
	
	iStartCase : INT;
	
	fbStartDelayExhFan : TON;
	fbStartDelaySupFan : TON;
	fbResetTon: TON;
	
	sTmpPv1 : STRING;
	sTmpPv2 : STRING;
	
	sRemainingTime : STRING;
	iRemainingTime : INT;
	
	bTmpStartSequenceFlag : BOOL; // internvariabel status startsekvens
	
	bExhDamperOutputInternal : BOOL; 
	bSupDamperOutputInternal : BOOL;
	
	bExhDamperOutputInternalTof : TOF; // Frånslagsfördröjning spjäll
	bSupDamperOutputInternalTof : TOF; // Frånslagsfördröjning spjäll
	fbAfterBlowElectricHeaterInternalTof : TOF; // Frånslagsfördröjning tilluftsfläkt vid efterblåsning elbatteri
	bAfterBlowElectricHeater : BOOL;
	
	fbServiceSwitchTOF : TOF;
	
	fbDrifttidsLarmTON : TON; // Larmar om aggregatet varit igång kontinuerligt utan driftstopp.
END_VAR
VAR PERSISTENT
	AD AT %M* : REAL := -1; //Larm om aggr. drifttid sedan senaste stopp > (-1 inaktiv. larm)~wp:[unit]timmar
END_VAR

//Drifttidslarm om aggregatet varit igång konstant i mer än inställd tid. 
mDrifttidslarm();
// Används för Adrians portlet i webport :)
PV9 := bFreezeAlarm OR bPumpAlarm OR bFireAlarm OR bSmokeAlarm OR bFuseAlarm OR bInterlock OR bInterlock2 OR bInterlock3 OR bCrosswiseInterlock;
fbInterlockAlarm(bInput:=bSupfanAlarm OR bExhfanAlarm , tAlarmDelay:= , bAutoReset:=FALSE , bAlarmOutput=> bCrosswiseInterlock);
bNormalOperation := (bTimechannel OR bExtendedOperation OR bUserDefinedOperation1 OR bUserDefinedOperation2) AND bSafeCon;
// Internvariabel för att blockera frånluftsfläkt vid nattanvärmning
bNightHeatingStatus := bNightHeating AND NOT bNormalOperation AND NOT bNightCooling AND bSafeCon;
fbNattAnvarmningsFtrig(CLK := bNightHeatingStatus);
fbNattAnvarmningsTof(IN:= fbNattAnvarmningsFtrig.Q,PT:=T#1S);
// Efterblåsning elbatteri
fbServiceSwitchTOF(IN:= NOT bServiceSwitch, PT:=tAfterblowStopDelay , Q=> , ET=> ); // För att köra efterblåsning vid serviceomkopplare
bStartConWithoutAfterblow := (bTimechannel OR bExtendedOperation OR bNightCooling OR bNightHeating OR bUserDefinedOperation1 OR bUserDefinedOperation2) AND bAfterblowActive AND NOT bFiredamperExercise;
fbAfterBlowElectricHeaterInternalTof(IN:= bStartConWithoutAfterblow , PT:=tAfterblowStopDelay , Q=>bAfterBlowElectricHeater , ET=> );
bAfterBlowElectricHeaterStatus := bAfterBlowElectricHeater AND ((NOT bNightHeating AND NOT bNormalOperation AND NOT bNightCooling) OR (fbServiceSwitchTOF.Q AND NOT fbServiceSwitchTOF.IN)) AND bSafeCon;

bStartCon := bSequenceStart AND (bTimechannel OR bExtendedOperation OR bNightCooling OR bNightHeating OR bUserDefinedOperation1 OR bUserDefinedOperation2 OR bAfterBlowElectricHeaterStatus) AND NOT bFiredamperExercise;
// Förregling samt handställningsförregling av fläktar. Kopplas till bSafe-ingång på fläkt
bSafeCon := NOT fbNattAnvarmningsTof.Q AND NOT bFreezeAlarm AND NOT bPumpAlarm AND NOT bFireAlarm AND NOT bSmokeAlarm AND NOT bFuseAlarm AND NOT bInterlock AND NOT bInterlock2 AND NOT bInterlock3 AND NOT bCrosswiseInterlock AND fbServiceSwitchTOF.Q;
(* Startsekvens - start *)
bExhDamperCon := (bStartCon AND bSafeCon);
(*************************** Utgång frånluftsspjäll ***************************)
bExhDamperOutputInternal := bExhDamperCon OR (bExhfan_M AND bExhfan_MCMD);
IF bNightHeatingStatus THEN
	fbStartDelayExhFan(IN:=bExhDamperCon , PT:=T#0S , Q=> , ET=> );
ELSE
	fbStartDelayExhFan(IN:=bExhDamperCon , PT:=tExhfanStartDelay , Q=> , ET=> );	
END_IF
(*************************** Utgång frånluftsfläkt ***************************)
bExhfanCon := fbStartDelayExhFan.Q AND (bStartCon AND bSafeCon);
bExhfanOutput := bExhfanCon AND NOT bNightHeatingStatus;
(*************************** Utgång tillluftsspjäll ***************************)
bSupDamperOutputInternal := (bExhfanCon AND (bStartCon AND bSafeCon)) OR (bSupfan_M AND bSupfan_MCMD);
fbStartDelaySupFan(IN:= bSupDamperOutputInternal , PT:=tSupfanStartDelay , Q=> , ET=> );
(*************************** Utgång frånluftsfläkt ***************************)
bSupfanOutput := fbStartDelaySupFan.Q AND (bStartCon AND bSafeCon);
(* Startsekvens - slut *)
bExhDamperOutputInternalTof(IN:=bExhDamperOutputInternal , PT:=tDamperStopDelay , Q=>bExhDamperOutput , ET=> );
bSupDamperOutputInternalTof(IN:= bSupDamperOutputInternal, PT:=tDamperStopDelay , Q=>bSupDamperOutput , ET=> );
//Status aggregatsdrift~wp:
IF bTimechannel AND bSafeCon THEN 
	sTmpPv1 := 'Normaldrift';
	bTmpStartSequenceFlag := TRUE;
ELSIF bExtendedOperation  AND bSafeCon THEN 
	sTmpPv1 := 'Forcerad drift';
	bTmpStartSequenceFlag := TRUE;
ELSIF bUserDefinedOperation1 AND bSafeCon THEN 
	sTmpPv1 := sUserDefinedOperation1;
	bTmpStartSequenceFlag := TRUE;
ELSIF bUserDefinedOperation2 AND bSafeCon THEN 
	sTmpPv1 := sUserDefinedOperation2;
	bTmpStartSequenceFlag := TRUE;
ELSIF bNightCooling  AND bSafeCon THEN
	sTmpPv1 := 'Nattkyla';
	bTmpStartSequenceFlag := TRUE;
ELSIF bNightHeating AND bSafeCon THEN
	sTmpPv1 := 'Nattanvärmning';
	bTmpStartSequenceFlag := TRUE;
ELSIF bAfterBlowElectricHeater AND bSafeCon THEN
	sTmpPv1 := 'Efterblåsning elbatteri';
	bTmpStartSequenceFlag := TRUE;
ELSE
 	sTmpPv1 := 'Aggregat stoppat';
	bTmpStartSequenceFlag := FALSE;
END_IF
IF NOT fbStartDelayExhFan.Q AND bTmpStartSequenceFlag AND NOT bNightHeating THEN
	sTmpPv1 := CONCAT(sTmpPv1, ', Startar frånluftsfläkt om ');
	iRemainingTime := TIME_TO_INT((fbStartDelayExhFan.PT -  fbStartDelayExhFan.ET)/ 1000);
	sRemainingTime := INT_TO_STRING(iRemainingTime);
	sRemainingTime := CONCAT(sRemainingTime, 's');
	sTmpPv1 := CONCAT(sTmpPv1, sRemainingTime);
ELSIF NOT fbStartDelaySupFan.Q AND bTmpStartSequenceFlag THEN
	sTmpPv1 := CONCAT(sTmpPv1, ', Startar tilluftsfläkt om ');	
	iRemainingTime := TIME_TO_INT((fbStartDelaySupFan.PT -  fbStartDelaySupFan.ET)/ 1000);
	sRemainingTime := INT_TO_STRING(iRemainingTime);
	sRemainingTime := CONCAT(sRemainingTime, 's');
	sTmpPv1 := CONCAT(sTmpPv1, sRemainingTime);
ELSIF bAfterBlowElectricHeater AND bTmpStartSequenceFlag AND NOT fbAfterBlowElectricHeaterInternalTof.IN THEN
	sTmpPv1 := CONCAT(sTmpPv1, ', Fläktar stannar stannar om ');	
	iRemainingTime := TIME_TO_INT((fbAfterBlowElectricHeaterInternalTof.PT -  fbAfterBlowElectricHeaterInternalTof.ET)/ 1000);
	sRemainingTime := INT_TO_STRING(iRemainingTime);
	sRemainingTime := CONCAT(sRemainingTime, 's');
	sTmpPv1 := CONCAT(sTmpPv1, sRemainingTime);	
ELSIF  bExhDamperOutput AND NOT bExhDamperOutputInternal THEN
	sTmpPv1 := CONCAT(sTmpPv1, ', Spjäll stänger om ');	
	iRemainingTime := TIME_TO_INT((bExhDamperOutputInternalTof.PT -  bExhDamperOutputInternalTof.ET)/ 1000);
	sRemainingTime := INT_TO_STRING(iRemainingTime);
	sRemainingTime := CONCAT(sRemainingTime, 's');
	sTmpPv1 := CONCAT(sTmpPv1, sRemainingTime);
END_IF
IF bCoolRecycling THEN
	sTmpPv1 := CONCAT(sTmpPv1, ', kylåtervinning VVX aktiv');
ELSIF bDefrostingVvx THEN 
	sTmpPv1 := CONCAT(sTmpPv1, ', avfrostning VVX');
END_IF
PV1 := sTmpPv1;
sTmpPv2 := ' ';
IF NOT bSequenceStart THEN
	sTmpPv2 := 'Fördröjd sekvensuppstart vid uppstart av plc.';
ELSIF bFreezeAlarm THEN 
	sTmpPv2 := 'Utlöst frysvakt - Åtgärda felorsak och återställ sedan förr. med resetknapp!';
ELSIF bPumpAlarm THEN 
	sTmpPv2 := 'Driftfel pump - Åtgärda felorsak och återställ sedan förr. med resetknapp!';
ELSIF bFireAlarm THEN
	sTmpPv2 := 'Utlöst brandlarm';
ELSIF bSmokeAlarm THEN
	sTmpPv2 := 'Utlöst rökdetektor';
ELSIF bFuseAlarm THEN
	sTmpPv2 := 'Utlöst automatsäkring';
ELSIF bInterlock THEN
	sTmpPv2 := sInterlockDescription;
ELSIF bInterlock2 THEN
	sTmpPv2 := sInterlock2Description;
ELSIF bInterlock3 THEN
	sTmpPv2 := sInterlock3Description;
ELSIF bCrosswiseInterlock THEN
	sTmpPv2 := 'Korsvis förregling - Åtgärda felorsak och återställ sedan förr. med resetknapp!';
ELSIF bServiceSwitch THEN
	sTmpPv2 := 'Serviceomkopplare ej i läge auto';
ELSIF bFiredamperExercise THEN
	sTmpPv2 := 'Motionskörning brandspjäll';
END_IF
PV2 := sTmpPv2;

METHOD PRIVATE mDrifttidslarm
VAR_INPUT
END_VAR
VAR
	rTemporaryTime : REAL;
END_VAR
VAR
	tTime : TIME;
	rTime : REAL;
END_VAR
	IF AD < -1 THEN
		AD := -1;
	ELSIF AD > 47 THEN 
		AD := 1100; 
	END_IF;
	IF AD = -1 THEN
		rTemporaryTime := 0;
	ELSE
		rTemporaryTime := AD;
	END_IF
	
	fbDrifttidsLarmTON(IN:=bStartCon AND  (AD <> -1), PT:=fRealToHour(rTemporaryTime) , Q=>FAULT , ET=> );

	tTime := fbDrifttidsLarmTON.PT - fbDrifttidsLarmTON.ET;
	
	rTime := TIME_TO_REAL(tTime) / 3600;
	
	IF tTime > T#0S AND tTime < fbDrifttidsLarmTON.PT  THEN
 		PV4 := CONCAT('Larm om aggregatet fortsätter gå utan driftstopp i ytterligare: ',CONCAT(INT_TO_STRING(REAL_TO_INT(rTime)), ' timmar'));
	ELSE
		PV4 := ' ';
	END_IF
END_METHOD

END_FUNCTION_BLOCK

// oaksLibrary/fbNightheating
(*
	Nattanvärmning Vinter
	Följande villkor behöver uppfyllas för att nattanvärmning ska aktiveras:
	- Rumstemperatur är lägre än inställt värde.
	- Utetemperatur är lägre än 10°C.
	Nattanvärmning stoppas om:
	- Rumstemperatur  överstiger inställt värde med 1°C.
	
	
 	V-tagg i detta block knyts till inputen bNightCooling i fbVentilationUnit.
*)
FUNCTION_BLOCK fbNightheating
VAR_INPUT
	rOutdoorTemp : ANY; // Utetemperatur Knyter man inget här används oaksGVL.rOutdoortemp
	rRoomTemp : REAL; // Rumstemperatur
	bDay : BOOL; // Tidkanal eller förlängd drift (knyt outputen bNormalOperation från fbVentilationUnit)
	bEnable : BOOL; // Knyt eventuell nattkyletidkanal hit
END_VAR
VAR_OUTPUT
	{attribute 'OPC.UA.DA' := '1'}
	PV4 AT %M*  : BOOL; //Driftvillkor utetemperatur~wp:[trendoptions]i:14400, t:1
	{attribute 'OPC.UA.DA' := '1'}
	PV5 AT %M*  : BOOL; //Driftvillkor rumstemperatur~wp:[trendoptions]i:14400, t:1
	{attribute 'OPC.UA.DA' := '1'}
	V	AT %M*  : BOOL; //Driftvillkor Nattanvärmning~wp:[trendoptions]i:14400, t:1
END_VAR
VAR
	rTempUsed : REAL; // Uteluftstemperatur
	fbRoomTempTON,fbOutdoorTempTON : TON;
END_VAR
VAR_INPUT PERSISTENT
	{attribute 'OPC.UA.DA' := '1'}
	SP1 AT %M* : REAL := 15; //Tillåt start av nattanvärmning om rumstemperatur underskrider~wp:[unit]°C[format]0.0
	{attribute 'OPC.UA.DA' := '1'}
	SP2 AT %M* : REAL := 10; //Tillåt nattanvärmning om utetemp underskrider~wp:[unit]°C[format]0.0
END_VAR



rTempUsed := F_GetTempToUse(rOutdoorTemp);

fbOutdoorTempTON.PT:=T#1M;
IF rTempUsed < SP2 THEN
	fbOutdoorTempTON.IN:= TRUE;
ELSIF rTempUsed > SP2 + 1 THEN
	fbOutdoorTempTON.IN:= FALSE;
END_IF;
fbOutdoorTempTON(Q=> PV4);

fbRoomTempTON.PT:=T#1M;
IF rRoomTemp < SP1 THEN
	fbRoomTempTON.IN:= TRUE;
ELSIF rRoomTemp > SP1 + 1  THEN
	fbRoomTempTON.IN:= FALSE;
END_IF;
fbRoomTempTON(Q=> PV5);

V := PV4 AND PV5 AND NOT bDay AND bEnable;

END_FUNCTION_BLOCK

// oaksLibrary/fbPresenceDetector
//Oaks AB
//2021-09-08
//Funktionsblock för digital närvarodetektor. Vid aktiv signal fördröjs frånslag med inställd tid. 
FUNCTION_BLOCK fbPresenceDetector
VAR_INPUT
	{attribute 'OPC.UA.DA' := '1'}
	V3 AT %I* : BOOL := FALSE; //Ingång närvarodetektor~wp:
	bInputInvert : BOOL := FALSE; //Invetering av ingång. False=NO (Slutande kontakt vid närvaro).
END_VAR

VAR_OUTPUT
	{attribute 'OPC.UA.DA' := '1'}
	PV1 AT %M* : REAL := 0; //Återstående närvarotid~wp:[unit]min[format]0
	{attribute 'OPC.UA.DA' := '1'}
	PV8 AT %M* : STRING := ' '; //Konfiguration digital ingång~wp:
	{attribute 'OPC.UA.DA' := '1'}
	V AT %M* : BOOL := FALSE; //Närvaro~wp:
END_VAR

VAR
	bInternalIndication : BOOL := FALSE;
	TOF_StopDelay : TOF;
	dTemp : DINT;
	
END_VAR

VAR_INPUT PERSISTENT
	{attribute 'OPC.UA.DA' := '1'}
	SP1 AT %M* : REAL := 60; //Närvarotid~wp:[unit]minuter[format]0
END_VAR

	//Invertering av ingång
	IF NOT bInputInvert THEN
		bInternalIndication :=  V3;
	ELSE
		bInternalIndication := NOT V3;
	END_IF
	
	//Frånslagsfördröjning
	TOF_StopDelay(IN:= bInternalIndication, PT:= fRealToMinute(SP1), Q=> V, ET=> );
	
	//Återstående timertid
	IF V THEN
		PV1 := DINT_TO_REAL((TIME_TO_DINT(TOF_StopDelay.PT) - TIME_TO_DINT(TOF_StopDelay.ET)) / 60000);
	ELSE 
		PV1 := 0;
	END_IF
		
	//Konfigurering ingång
	IF bInputInvert THEN
			PV8 := 'NC (Brytande kontakt vid närvaro)'; 
	ELSIF NOT bInputInvert THEN 
			PV8 := 'NO (Slutande kontakt vid närvaro)';
	END_IF

END_FUNCTION_BLOCK

// oaksLibrary/fbResetButton
// Resetknapp för knytning till io. Går även att resetta genom tagglista genom att sätta M till 1.
// CMD knyts internt i de block som ej är autoresettande. 
FUNCTION_BLOCK fbResetButton
VAR
	{attribute 'OPC.UA.DA' := '1'}
	V  AT %I*: BOOL; //Ingång resetknapp~wp:[trendoptions]i:14400, t:1
	{attribute 'OPC.UA.DA' := '1'}

	fbResetTon : TON;
	fbResetTonRst : TON;
	
	fbAlarmResetButton : fbAlarm;
	
	{attribute 'OPC.UA.DA' := '1'}
	M AT %M* : BOOL; //Handställning (används för återställning från webport)~wp:[trendoptions]i:14400, t:1
	RST AT %M* : BOOL; //Handställning (används för återställning från webport)~wp:[trendoptions]i:14400, t:1
END_VAR
VAR_OUTPUT
	CMD AT %M* : BOOL; //Aktivt larm som kräver manuell kvittering för återställning~wp:[trendoptions]i:14400, t:1
	CMD1 AT %M* : BOOL; //Aktivt larm (både de som kräver och inte kräver manuell kvittering för återställning)~wp:[trendoptions]i:14400, t:1
	FAULT AT %M* : BOOL; //Resetknapp på apparatskåpsfront har varit intryckt under lång tid~wp:
END_VAR

	oaksGVL.bReset := V OR M OR RST;

	// Sätter återställning av M till FALSE efter 5 sekunder
	IF M THEN
		fbResetTon.IN := TRUE;
		IF fbResetTon.Q THEN
			M := FALSE;
		END_IF
	ELSE
		fbResetTon.IN := FALSE;
	END_IF
	fbResetTon.PT := T#5S;
	fbResetTon();
	
	// Sätter återställning av RST till FALSE efter 5 sekunder
	IF RST THEN
		fbResetTonRst.IN := TRUE;
		IF fbResetTonRst.Q THEN
			RST := FALSE;
		END_IF
	ELSE
		fbResetTonRst.IN := FALSE;
	END_IF
	fbResetTonRst.PT := T#5S;
	fbResetTonRst();
	
	CMD := oaksgvl.bSummalarmEjAutoReset;
	CMD1 := oaksgvl.bSummalarm;
	
	fbAlarmResetButton(bInput:=V , tAlarmDelay:=T#1m , bAutoReset:=true , bAlarmOutput=>FAULT );

END_FUNCTION_BLOCK

// oaksLibrary/fbServiceSwitch
// Serviceomkopplare med larm
FUNCTION_BLOCK fbServiceSwitch
VAR_INPUT
	bInvert : BOOL; // Invertering av io-ingång för larm
	bInvertIndication : BOOL; // Inverterar indikering (V-tagg)
END_VAR
VAR
	{attribute 'OPC.UA.DA' := '1'}
	PV4 AT %I* : BOOL; //Läge serviceomkopplare~wp:[trendoptions]i:14400, t:1
	bStartSignal : BOOL; 
END_VAR
VAR_OUTPUT
	{attribute 'OPC.UA.DA' := '1'}
	V AT %M*: BOOL; //Utsignal för visning i webport~wp:[trendoptions]i:14400, t:1
	{attribute 'OPC.UA.DA' := '1'}
	CMD AT %M*: BOOL; //Utsignal~wp:[trendoptions]i:14400, t:1
	{attribute 'OPC.UA.DA' := '1'}
	AL AT %M*: BOOL; //Omkopplare ej i läge auto~wp:
	{attribute 'OPC.UA.DA' := '1'}
	AL8 AT %M*: BOOL; //Utsignal handställd~wp:[alarmoptions]p:3
END_VAR
VAR
	fbAlarm1 : fbAlarm;
END_VAR
VAR_INPUT PERSISTENT
	{attribute 'OPC.UA.DA' := '1'}
	M AT %M*: BOOL; //Handställning~wp:[trendoptions]i:14400, t:1
	{attribute 'OPC.UA.DA' := '1'}
	MCMD AT %M*: BOOL; //Styrsignal handställning~wp:[trendoptions]i:14400, t:1
END_VAR



	fbAlarm1(
	bInput:= CMD, 
	tAlarmDelay:= , 
	bAutoReset:= TRUE, 
	bAlarmOutput=>AL );
	
	
	AL8 := M;
	

	bStartSignal :=  (NOT PV4 AND NOT M) OR (M AND MCMD);
		
	
	
	IF bInvert THEN
		CMD := NOT bStartSignal;
	ELSE
		CMD :=  bStartSignal;
	END_IF
	
	
	IF NOT bInvertIndication THEN 
		V := NOT CMD;
	ELSE
		V := CMD;
	END_IF

END_FUNCTION_BLOCK

// oaksLibrary/fbServiceSwitch01A
//Oaks AB
//2020-09-28
//Funktionsblock för serviceomkopplare för 0-1-AUTO. Indikering på både Auto-läge och manuellt-läge samtidigt ger bError.
FUNCTION_BLOCK fbServiceSwitch01A
VAR_INPUT
	bInvertOn : BOOL := FALSE; //Invertering ingång till (Signal går till vid aktivering = FALSE)
	bInvertAuto : BOOL := FALSE; //Invertering ingång auto (Signal går till vid aktivering = FALSE)
	{attribute 'OPC.UA.DA' := '1'}
	V3 AT %I* : BOOL; //Ingång omkopplare till~wp:[trendoptions]i:14400, t:1
	{attribute 'OPC.UA.DA' := '1'}
	V4 AT %I* : BOOL; //Ingång omkoppalre auto~wp:[trendoptions]i:14400, t:1
END_VAR
VAR
	bOnInternal : BOOL;
	bAutoInternal : BOOL;
	fbAlarm1: fbAlarm;
	
END_VAR
VAR_OUTPUT
	{attribute 'OPC.UA.DA' := '1'}
	PV AT %M*: STRING; //Utsignal för visning i webport~wp:[trendoptions]i:14400, t:1
	{attribute 'OPC.UA.DA' := '1'}
	V AT %M*: INT; //Driftläge Av(0)/Till(1)/Auto(2)~wp:[trendoptions]i:14400, t:1
	{attribute 'OPC.UA.DA' := '1'}
	AL AT %M*: BOOL; //Omkopplare ej i läge Auto~wp:
	bOff : BOOL; //Av (TRUE om varken Auto eller Till är aktiv på omkopplare)
	bOn : BOOL; //Till (TRUE om Till är aktivt på omkopplare)
	bAuto : BOOL; //Auto (TRUE om Auto är aktivt på omkopplare)
	bError : BOOL; //Fel konfiguration (Auto och Till är aktiva samtidigt)
	
END_VAR

VAR_INPUT PERSISTENT
	//M AT %M*: BOOL; //Handställning~wp:[trendoptions]i:300
	//MCMD AT %M*: BOOL; //Styrsignal handställning~wp:[trendoptions]i:300
END_VAR

	//Invertering ingång manuellt-läge
	IF bInvertOn THEN
		bOnInternal := NOT V3;
	ELSE
		bOnInternal := V3;
	END_IF
		
	//Invertering ingång auto-läge
	IF bInvertAuto THEN
		bAutoInternal := NOT V4;
	ELSE
		bAutoInternal := V4;
	END_IF
	
	//Konfigurationskoll
	bError := (bOnInternal AND bAutoInternal);
	
	//Larm ej i auto
	fbAlarm1(
	bInput:= NOT bAutoInternal AND NOT bError, 
	tAlarmDelay:= T#5S, 
	bAutoReset:= TRUE, 
	bAlarmOutput=>AL );
			
	//Driftläge
	IF bError THEN
		PV := 'Fel IO-konfiguration';
		V := 0; //Av
		bOff := TRUE;
		bOn := FALSE;
		bAuto := FALSE;
	ELSIF NOT bOnInternal AND NOT bAutoInternal THEN
		PV := 'Av';
		V := 0; //Av
		bOff := TRUE;
		bOn := FALSE;
		bAuto := FALSE;
	ELSIF bOnInternal THEN
		PV := 'Till';
		V := 1; //Till
		bOff := FALSE;
		bOn := TRUE;
		bAuto := FALSE;
	ELSIF bAutoInternal THEN
		PV := 'Auto';
		V := 2; //Auto
		bOff := FALSE;
		bOn := FALSE;
		bAuto := TRUE;
	END_IF

END_FUNCTION_BLOCK

// oaksLibrary/fbTimeChannelWp
FUNCTION_BLOCK fbTimeChannelWp
VAR_INPUT
	iWatchdogConfig : INT := 1; //Välj vilket läge tidkanal ska vara i vid komm-fel mot webport. -1 om senaste läge önskas.
	
END_VAR
VAR
	{attribute 'OPC.UA.DA' := '1'}
	V AT %M*  : INT; //Indikering för visning i webport~wp:[trendoptions]i:14400, t:1
END_VAR
VAR_OUTPUT
	bStart : BOOL; // Till om CMD > 0
END_VAR
VAR_OUTPUT PERSISTENT
	{attribute 'OPC.UA.DA' := '1'}
	CMD AT %M*  : INT; //Utsignal~wp:[trendoptions]i:14400, t:1
END_VAR

IF oaksGVL.bWatchdog AND iWatchdogConfig <> -1 THEN
	CMD := iWatchdogConfig;
END_IF

bStart :=CMD > 0;
V := CMD;

END_FUNCTION_BLOCK

// oaksLibrary/fbWatchdogSwitching
//Funktionsblock för Watchdog funktion. Då växling uteblir på V3 under 60 sekunder utgår watchdog-larm.
FUNCTION_BLOCK fbWatchdogSwitching
VAR_OUTPUT
	FAULT AT %M* : BOOL; //Utlöst watchdog~wp:
END_VAR
VAR
	{attribute 'OPC.UA.DA' := '1'}
	V3 AT %M* : BOOL; //Växlande indikering~wp:
	timer01 : ton;
	timer02 : ton;
	fbAlarm: fbAlarm;
END_VAR

timer01(IN:= NOT V3, PT:=T#900S , Q=> , ET=> );
timer02(IN:= V3, PT:=T#900S , Q=> , ET=> );

fbAlarm(bInput:= timer01.Q OR timer02.Q, tAlarmDelay:= T#1S, bAutoReset:= TRUE, bAlarmOutput=>FAULT);

oaksgvl.bWatchdog := FAULT;

END_FUNCTION_BLOCK
